PROGRAM PRG_LVCP1
VAR
END_VAR

	PRG_LVCP1_PowerMeasurement();	

	PRG_LVCP1_CompensationCalculate();

	PRG_LVCP1_MainDisconnector();
	
	PRG_Lvcp1_Colors();
	
	PRG_LVCP1_Group1();
	
	PRG_LVCP1_Group2();
	
	PRG_LVCP1_Group3();	
	
	PRG_LVCP1_Group4();	

	PRG_LVCP1_Group5();	

	PRG_LVCP1_Group6();	

	PRG_LVCP1_Group7();	

	PRG_LVCP1_Group8();	

	PRG_LVCP1_Group9();	

	PRG_LVCP1_Group10();

END_PROGRAM

(* stored: Version 1.1.0.1, ProductVersion 3.1.4024.14
   POU PRG_LVCP1: Id {0304955c-4377-4d31-9ad2-31d77e8321af}, SpecialFunc None *)
